TYPE stOPCUASkill :
STRUCT
	Start: BOOL;
	Cancel: BOOL;
	Reset: BOOL;
	Ready: BOOL;
	Busy: BOOL;
	Done: BOOL;
	Success: BOOL;
	Error: BOOL;
	Result: STRING;
	ErrorCode: UINT;
	ErrorMessage: STRING;
	State: UINT;
	Progress: REAL;
	Timeout: REAL;
	RequestID: UINT;
	ResultRequestID: UINT;
	Timestamp: TIME;
	
END_STRUCT
END_TYPE

(* stored: Version 1.1.0.1, ProductVersion 3.1.4026.18
   DUT stOPCUASkill: Id {0deeb3e2-3419-4505-81b8-79b38cbf2e27} *)
